FUNCTION_BLOCK FB_SavePersistentData
VAR_INPUT
END_VAR
VAR_OUTPUT
END_VAR
VAR
	instFbClkPrgWritePersistentData: CLK_PRG;
	instFbWritePersistentData: FB_WritePersistentData;
	savePersisteData: BOOL;
	cpuPowerFailDetected: BOOL;
	writePersistentDataBusy: BOOL;
	writePersistentDataErr: BOOL;
	saveCounter: DINT;
	instFBSUpsBapi: FB_S_UPS_BAPI;
	
	writePersistentDataErrId :UDINT;
END_VAR
VAR // added by the converter: edge detectors and wires of the graphical bodies
    _w1 : DINT;
END_VAR

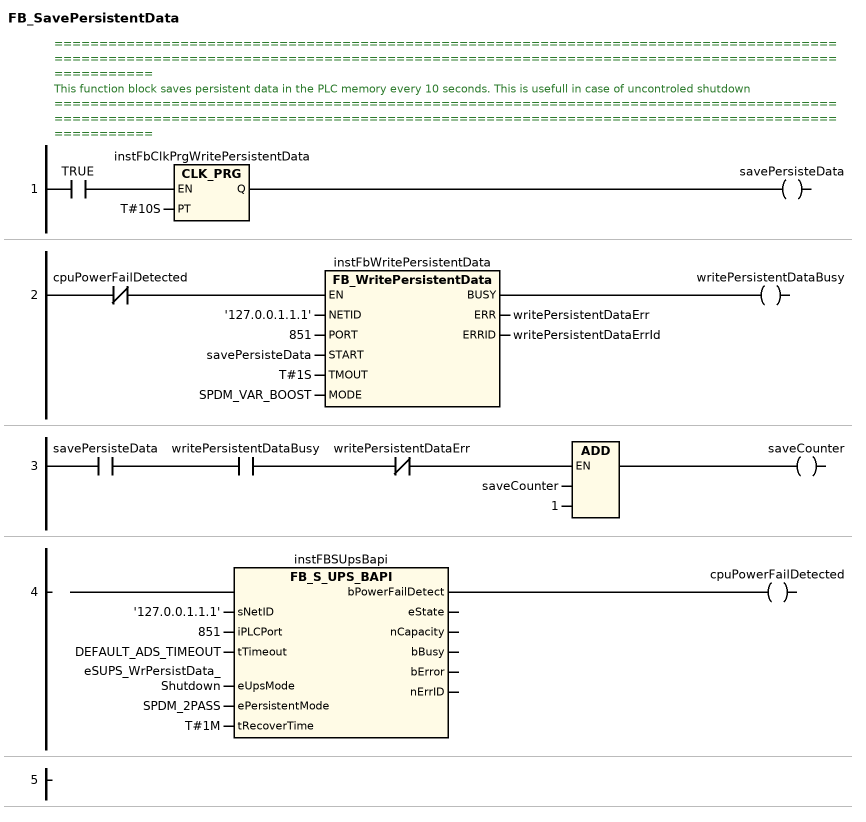
// NETWORK 1
// 					=========================================================================================================================================================================================
//
// This function block saves persistent data in the PLC memory every 10 seconds. This is usefull in case of uncontroled shutdown
//
// =========================================================================================================================================================================================
//
instFbClkPrgWritePersistentData(PT := T#10S); // CLK_PRG
savePersisteData := instFbClkPrgWritePersistentData.Q;

// NETWORK 2
IF NOT cpuPowerFailDetected THEN
    instFbWritePersistentData(
        NETID := '127.0.0.1.1.1',
        PORT := 851,
        START := savePersisteData,
        TMOUT := T#1S,
        MODE := SPDM_VAR_BOOST,
        ERR => writePersistentDataErr,
        ERRID => writePersistentDataErrId); // FB_WritePersistentData
END_IF
writePersistentDataBusy := instFbWritePersistentData.BUSY;

// NETWORK 3
IF savePersisteData AND writePersistentDataBusy AND NOT writePersistentDataErr THEN _w1 := saveCounter + 1; END_IF
saveCounter := _w1;

// NETWORK 4
instFBSUpsBapi(
    sNetID := '127.0.0.1.1.1',
    iPLCPort := 851,
    tTimeout := DEFAULT_ADS_TIMEOUT,
    eUpsMode := eSUPS_WrPersistData_Shutdown,
    ePersistentMode := SPDM_2PASS,
    tRecoverTime := T#1M); // FB_S_UPS_BAPI
cpuPowerFailDetected := instFBSUpsBapi.bPowerFailDetect;

// NETWORK 5

END_FUNCTION_BLOCK

(* stored: Version 1.1.0.1, ProductVersion 3.1.4024.15
   POU FB_SavePersistentData: Id {0b4790df-99db-0804-1ed4-5a7679196a3c}, SpecialFunc None *)
